FUNCTION_BLOCK TOffTimer
VAR
    TOF1 : TOF;
END_VAR

METHOD Delay : BOOL
VAR_INPUT
    In : BOOL;
END_VAR
TOF1(IN := In);
Delay := TOF1.Q;
END_METHOD

METHOD FB_init : BOOL
VAR_INPUT
	bInitRetains : BOOL; // if TRUE, the retain variables are initialized (warm start / cold start)
	bInCopyCode : BOOL;  // if TRUE, the instance afterwards gets moved into the copy code (online change)
    PresetTime : LREAL; // seconds
END_VAR
TOF1.PT := LREAL_TO_TIME(PresetTime * 1000);
END_METHOD

PROPERTY OutputState : BOOL
GET
OutputState := TOF1.Q;
END_GET
END_PROPERTY

PROPERTY PresetTime : LREAL
GET
PresetTime := TIME_TO_LREAL(TOF1.PT)/1000.0; // in seconds
END_GET
SET
TOF1.PT := LREAL_TO_TIME(PresetTime * 1000);
END_SET
END_PROPERTY

END_FUNCTION_BLOCK

(* stored: Version 1.1.0.1, ProductVersion 3.1.4024.3
   POU TOffTimer: Id {eebce3f3-8192-4720-b0f0-7d130b8b7e89}, SpecialFunc None
   Method Delay: Id {4bdaf898-afaa-464d-a527-f1288374e158}
   Method FB_init: Id {95bab69f-9f7e-4f08-83da-293496638899}
   Property OutputState: Id {c1fdc1b8-386e-46d1-a827-bfdbd19fce8e}
   Get Get: Id {e9e8c2e6-68a4-4de3-bd76-22d823c7ac0e}
   Property PresetTime: Id {22180b71-8abb-4e5e-b1cf-e8153537742b}
   Get Get: Id {a427294d-f691-4c0b-b912-7b7ab0d94528}
   Set Set: Id {fe00e5b0-3cbe-42ff-abf8-f5ec69ac516f} *)
